# EPICS substitutions: apps/mpodLvApp/Db/subs/fttrklv.substitutions
file "db/mpod8008l.db" {
    pattern {HOST,CH,SCAN,PORT,DETALIAS}
{"%(fttlv)","0","2 second","B_HW_FTTLV_Sl0_Ch0","B_DET_FTT_LV_0"}
{"%(fttlv)","1","2 second","B_HW_FTTLV_Sl0_Ch1","B_DET_FTT_LV_1"}
{"%(fttlv)","2","2 second","B_HW_FTTLV_Sl0_Ch2","B_DET_FTT_LV_2"}
}
